// TwinCAT 3 PLC project TcUnitVerifier
// Title: TcUnit verifier
// Company: www.tcunit.org
// Author: Jakob Sagatowski and contributors
// ProjectVersion: 1.2.1.0
// Description: This project is can be used to verify the different functions of TcUnit. It has various test suites to test different functions in TcUnit. By making sure to comment out everything except the test suite that is interesting it is possible to test only the specific function of TcUnit that is interesting.
// ProgramVersion: 3.1.4026.21
// libraries:
//   SysDir, * (System)
//   SysFile, * (System)
//   Tc2_Standard, * (Beckhoff Automation GmbH)
//   Tc2_System, * (Beckhoff Automation GmbH)
//   Tc3_Module, * (Beckhoff Automation GmbH)
//   TcUnit, * (www.tcunit.org)
//   Base Interfaces,newest,System
// project tree:
//   / PlcTask.TcTTO (not stored)
//   POUs/ FB_ProtectedVariables.TcPOU (not stored)
//   Test/ FB_AdjustAssertFailureMessageToMax253CharLengthTest.TcPOU (not stored), FB_TestDurationMeasurement.TcPOU (not stored), FB_AnyPrimitiveTypes.TcPOU (not stored), FB_AnyToUnionValue.TcPOU (not stored), FB_ArrayPrimitiveTypes.TcPOU (not stored), FB_AssertCountExceedsMaxNumber.TcPOU (not stored), FB_AssertEveryFailedTestTwice.TcPOU (not stored), FB_AssertEveryFailedTestTwiceArrayVersion.TcPOU (not stored), FB_AssertTrueFalse.TcPOU (not stored), FB_CheckIfSpecificTestIsFinished.TcPOU (not stored), FB_CreateDisabledTest.TcPOU (not stored), FB_CreateFourTestsWithSameName.TcPOU (not stored), FB_EmptyAssertionMessage.TcPOU (not stored), FB_EmptyTestSuite.TcPOU (not stored), FB_ExtendedTestInformation.TcPOU (not stored), FB_MultipleAssertWithSameParametersInDifferentCyclesAndInSameTest.TcPOU (not stored), FB_MultipleAssertWithSameParametersInDifferentCyclesButWithDifferentTests.TcPOU (not stored), FB_MultipleAssertWithSameParametersInSameCycleWithSameTest.TcPOU (not stored), FB_SkipAssertionsWhenFinished.TcPOU (not stored), FB_PrimitiveTypes.TcPOU (not stored), FB_TestFileControl.TcPOU (not stored), FB_TestFinishedNamed.TcPOU (not stored), FB_TestNumberOfAssertionsCalculation.TcPOU (not stored), FB_TestStreamBuffer.TcPOU (not stored), FB_TestXmlControl.TcPOU (not stored), FB_WriteProtectedFunctions.TcPOU (not stored), FB_TestFinishedNamedDoesNotExist.TcPOU (not stored), PRG_TEST.TcPOU (not stored), FB_SequentialSingleSuite.TcPOU, PRG_TEST_SEQUENCE.TcPOU
//   Version/ Global_Version.TcGVL
// real-time tasks:
//   TASK PlcTask: cycle T#10ms, priority 20, ADS port 350

// ---- Version/Global_Version.TcGVL
{attribute 'TcGenerated'}
{attribute 'no-analysis'}
{attribute 'linkalways'}
// This function has been automatically generated from the project information.
VAR_GLOBAL CONSTANT
	{attribute 'const_non_replaced'}
	stLibVersion_TcUnit_verifier : ST_LibVersion := (iMajor := 1, iMinor := 2, iBuild := 1, iRevision := 0, sVersion := '1.2.1.0');
END_VAR

// ---- Test/FB_SequentialSingleSuite.TcPOU
// One passing test; used by PRG_TEST_SEQUENCE for the N=1 sequential check.
FUNCTION_BLOCK FB_SequentialSingleSuite EXTENDS TcUnit.FB_TestSuite

TEST('Test_SingleSequentialPass');
AssertTrue(Condition := TRUE, Message := 'Single-suite sequential run');
TEST_FINISHED();

END_FUNCTION_BLOCK

// ---- Test/PRG_TEST_SEQUENCE.TcPOU
(* Committed single-suite RUN_IN_SEQUENCE check (precursor of the fully
   automated sequential verifier configuration; see the Phase 5 verifier plan).
   Usage: exclude PRG_TEST from build, assign PlcTask to this PRG, run, and
   verify TcUnit.GVL_TcUnit.TcUnitRunner.AllTestSuitesFinished latches TRUE with
   TcUnit.GVL_TcUnit.NumberOfInitializedTestSuites = 1 (same empirical suite-count
   preflight as the step-0 campaigns).
   With exactly one registered suite, the 2026.7.17.1 baseline never latches (the
   final-suite branch never published the finished count); the Step-0 candidate
   latches. *)
PROGRAM PRG_TEST_SEQUENCE
VAR
    SingleSuite : FB_SequentialSingleSuite;
END_VAR

TcUnit.RUN_IN_SEQUENCE();

END_PROGRAM
